// TIA Portal V20 export
// export: Created 2025-12-01T14:57:01.5792042Z, ExportSetting None, DisplayName Totally Integrated Automation Portal, DisplayVersion V20 Update 3, DisplayName TIA Portal Openness, DisplayVersion V20 Update 3, DisplayName TIA Portal Version Control Interface, DisplayVersion V20 Update 3, DisplayName STEP 7 Professional, DisplayVersion V20 Update 3, DisplayName STEP 7 Safety, DisplayVersion V20 Update 2, DisplayName WinCC Basic/Comfort/Advanced, DisplayVersion V20 Update 3, DisplayName WinCC Professional, DisplayVersion V20 Update 3, DisplayName WinCC Unified, DisplayVersion V20 Update 3
FUNCTION "FC458_TL_EMP_E1_S2_AUS" : Void   // FC458, LAD
{ S7_Optimized_Access := 'FALSE' }
AUTHOR : TLigero
NAME : 20160208
VERSION : 3.5
// stored: AutoNumber false, SetENOAutomatically false
   VAR_INPUT
      Mesa : UInt;
      En_Tension : Bool;
      phsMx_E1 : Bool;
      Termico_E1_Tx : Bool;
      Avance_E1_Tx_Ok : Bool;
      En_Emp_Recogido : Bool;
      En_Emp_Extendido : Bool;
      AVTF_MAnt_Mx : Bool;
      PTF_Mx_MSig : Bool;
      NXT_Avance : Bool;
      V_CNT_ApHsMx_E1 : UDInt;
      V_Paro : UDInt;
      V_Emp_Sacado : UDInt;
      V_TOut_Empujador : UDInt;
      V_TOut_Tx_Mx : UDInt;
   END_VAR
   VAR_OUTPUT
      PTF_MAnt_Mx : Bool;
      AVTF_Mx_MSig : Bool;
      NXT_Descarga_Act : Bool;
   END_VAR
   VAR_IN_OUT
      Mem_Aux_FNE1 : Bool;
      Mem_FN_phs_E1 : Bool;
      Mem_Aux_FNS2 : Bool;
      Mem_FN_phs_S2 : Bool;
      Mem_Flanco_Recog : Bool;
   END_VAR
   VAR_TEMP
      Mem_CNT_Aus_Ent : Bool;
      Temp_Emp_Sacado : Bool;
      Aux_Parar : Bool;
      tout_atasco : Bool;
      Tout_Empujador : Bool;
      Mem_CNT_Tmp_Paro_Tx : Bool;
      TEMP_MA_TR_Pos_E1 : Bool;
      TEMP_MA_TR_Pos_S2 : Bool;
      ok_tension : Bool;
   END_VAR
   VAR_TEMP   // added for the SCL form of the ladder/FBD networks
      _w1 : Bool;
      _w2 : Bool;
   END_VAR
BEGIN

REGION Network 1: Marca General Error
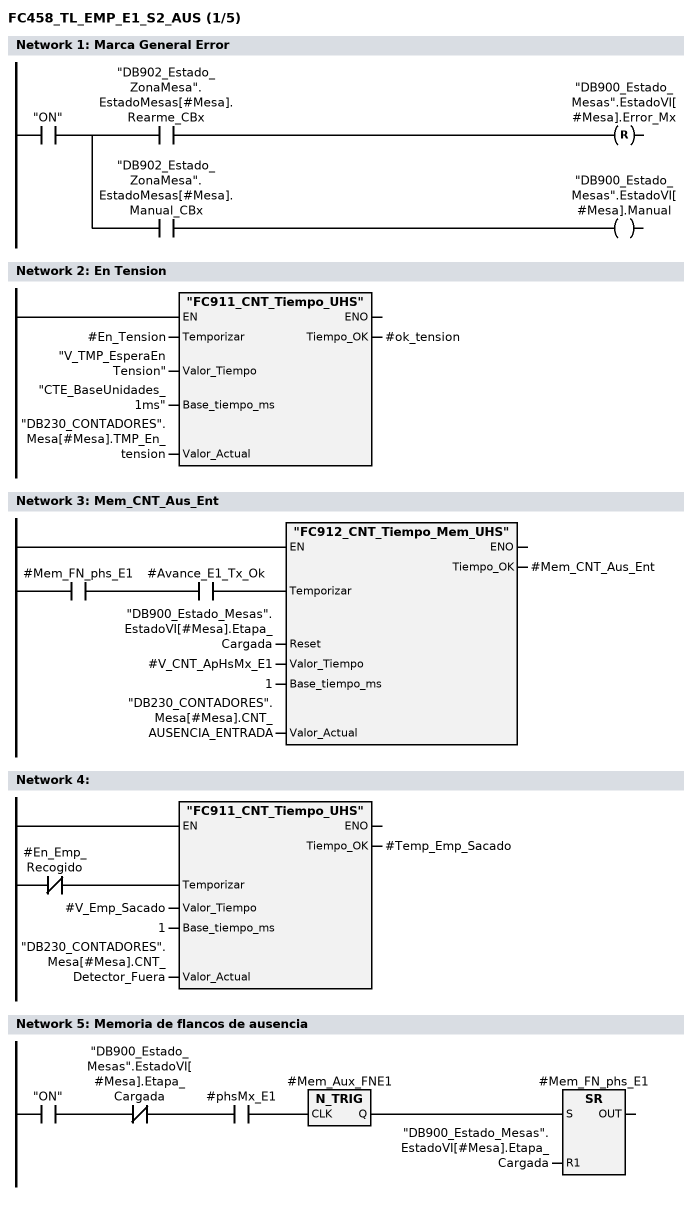
   RUNG wire#powerrail
      Contact( "ON" )
      wire#w1
      Contact( "DB902_Estado_ZonaMesa".EstadoMesas[#Mesa].Rearme_CBx )
      R_Coil( "DB900_Estado_Mesas".EstadoVI[#Mesa].Error_Mx )
   END_RUNG
   RUNG wire#w1
      Contact( "DB902_Estado_ZonaMesa".EstadoMesas[#Mesa].Manual_CBx )
      Coil( "DB900_Estado_Mesas".EstadoVI[#Mesa].Manual )
   END_RUNG
   // the same network as SCL:
   IF "ON" AND "DB902_Estado_ZonaMesa".EstadoMesas[#Mesa].Rearme_CBx THEN
       "DB900_Estado_Mesas".EstadoVI[#Mesa].Error_Mx := FALSE;
   END_IF;
   "DB900_Estado_Mesas".EstadoVI[#Mesa].Manual := "ON" AND "DB902_Estado_ZonaMesa".EstadoMesas[#Mesa].Manual_CBx;
END_REGION

REGION Network 2: En Tension
   RUNG wire#powerrail
      "FC911_CNT_Tiempo_UHS"(Temporizar := #En_Tension, Valor_Tiempo := "V_TMP_EsperaEnTension", Base_tiempo_ms := "CTE_BaseUnidades_1ms", Valor_Actual := "DB230_CONTADORES".Mesa[#Mesa].TMP_En_tension, Tiempo_OK => #ok_tension)
   END_RUNG
   // the same network as SCL:
   "FC911_CNT_Tiempo_UHS"(Temporizar := #En_Tension,
                          Valor_Tiempo := "V_TMP_EsperaEnTension",
                          Base_tiempo_ms := "CTE_BaseUnidades_1ms",
                          Valor_Actual := "DB230_CONTADORES".Mesa[#Mesa].TMP_En_tension,
                          Tiempo_OK => #ok_tension);
END_REGION

REGION Network 3: Mem_CNT_Aus_Ent
   RUNG wire#powerrail
      "FC912_CNT_Tiempo_Mem_UHS"(Temporizar := wire#w1, Reset := "DB900_Estado_Mesas".EstadoVI[#Mesa].Etapa_Cargada, Valor_Tiempo := #V_CNT_ApHsMx_E1, Base_tiempo_ms := 1, Valor_Actual := "DB230_CONTADORES".Mesa[#Mesa].CNT_AUSENCIA_ENTRADA, Tiempo_OK => #Mem_CNT_Aus_Ent)
   END_RUNG
   RUNG wire#powerrail
      Contact( #Mem_FN_phs_E1 )
      Contact( #Avance_E1_Tx_Ok )
   END_RUNG wire#w1
   // the same network as SCL:
   "FC912_CNT_Tiempo_Mem_UHS"(Temporizar := #Mem_FN_phs_E1 AND #Avance_E1_Tx_Ok,
                           Reset := "DB900_Estado_Mesas".EstadoVI[#Mesa].Etapa_Cargada,
                           Valor_Tiempo := #V_CNT_ApHsMx_E1,
                           Base_tiempo_ms := 1,
                           Valor_Actual := "DB230_CONTADORES".Mesa[#Mesa].CNT_AUSENCIA_ENTRADA,
                           Tiempo_OK => #Mem_CNT_Aus_Ent);
END_REGION

REGION Network 4
   RUNG wire#powerrail
      "FC911_CNT_Tiempo_UHS"(Temporizar := wire#w1, Valor_Tiempo := #V_Emp_Sacado, Base_tiempo_ms := 1, Valor_Actual := "DB230_CONTADORES".Mesa[#Mesa].CNT_Detector_Fuera, Tiempo_OK => #Temp_Emp_Sacado)
   END_RUNG
   RUNG wire#powerrail
      I_Contact( #En_Emp_Recogido )
   END_RUNG wire#w1
   // the same network as SCL:
   "FC911_CNT_Tiempo_UHS"(Temporizar := NOT #En_Emp_Recogido,
                          Valor_Tiempo := #V_Emp_Sacado,
                          Base_tiempo_ms := 1,
                          Valor_Actual := "DB230_CONTADORES".Mesa[#Mesa].CNT_Detector_Fuera,
                          Tiempo_OK => #Temp_Emp_Sacado);
END_REGION

REGION Network 5: Memoria de flancos de ausencia
   RUNG wire#powerrail
      Contact( "ON" )
      I_Contact( "DB900_Estado_Mesas".EstadoVI[#Mesa].Etapa_Cargada )
      Contact( #phsMx_E1 )
      N_Trig( #Mem_Aux_FNE1 )
      S_SR(operand := #Mem_FN_phs_E1, r1 := "DB900_Estado_Mesas".EstadoVI[#Mesa].Etapa_Cargada)
   END_RUNG
   // the same network as SCL:
   #_w1 := "ON" AND NOT "DB900_Estado_Mesas".EstadoVI[#Mesa].Etapa_Cargada AND #phsMx_E1;
   #_w2 := NOT #_w1 AND #Mem_Aux_FNE1;   // falling edge
   #Mem_Aux_FNE1 := #_w1;
   IF #_w2 THEN
       #Mem_FN_phs_E1 := TRUE;   // SR flip-flop
   END_IF;
   IF "DB900_Estado_Mesas".EstadoVI[#Mesa].Etapa_Cargada THEN #Mem_FN_phs_E1 := FALSE; END_IF;
END_REGION

REGION Network 6: PARO
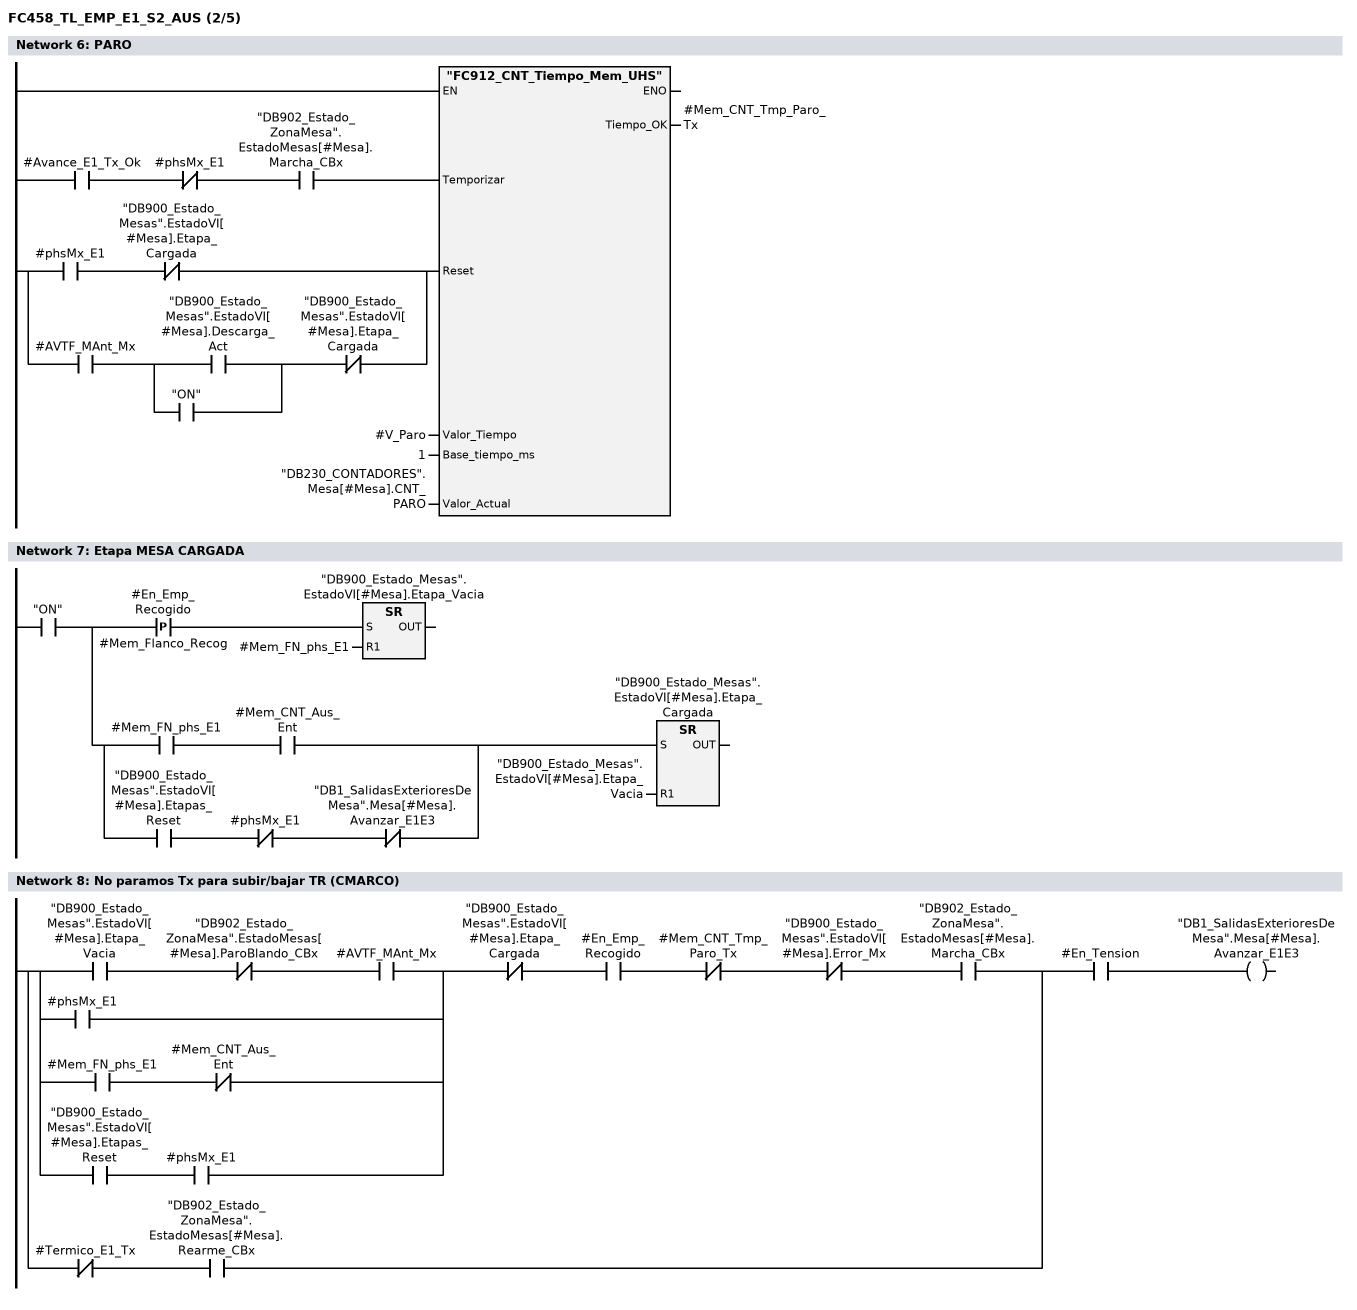
   RUNG wire#powerrail
      "FC912_CNT_Tiempo_Mem_UHS"(Temporizar := wire#w1, Reset := wire#w4, Valor_Tiempo := #V_Paro, Base_tiempo_ms := 1, Valor_Actual := "DB230_CONTADORES".Mesa[#Mesa].CNT_PARO, Tiempo_OK => #Mem_CNT_Tmp_Paro_Tx)
   END_RUNG
   RUNG wire#powerrail
      Contact( #Avance_E1_Tx_Ok )
      I_Contact( #phsMx_E1 )
      Contact( "DB902_Estado_ZonaMesa".EstadoMesas[#Mesa].Marcha_CBx )
   END_RUNG wire#w1
   RUNG wire#powerrail
      Contact( #phsMx_E1 )
      I_Contact( "DB900_Estado_Mesas".EstadoVI[#Mesa].Etapa_Cargada )
   END_RUNG wire#w4
   RUNG wire#powerrail
      Contact( #AVTF_MAnt_Mx )
      wire#w2
      Contact( "DB900_Estado_Mesas".EstadoVI[#Mesa].Descarga_Act )
      wire#w3
      I_Contact( "DB900_Estado_Mesas".EstadoVI[#Mesa].Etapa_Cargada )
   END_RUNG wire#w4
   RUNG wire#w2
      Contact( "ON" )
   END_RUNG wire#w3
   // the same network as SCL:
   "FC912_CNT_Tiempo_Mem_UHS"(Temporizar := #Avance_E1_Tx_Ok AND NOT #phsMx_E1 AND "DB902_Estado_ZonaMesa".EstadoMesas[#Mesa].Marcha_CBx,
                           Reset := (#phsMx_E1 AND NOT "DB900_Estado_Mesas".EstadoVI[#Mesa].Etapa_Cargada) OR (#AVTF_MAnt_Mx AND ("DB900_Estado_Mesas".EstadoVI[#Mesa].Descarga_Act OR "ON") AND NOT "DB900_Estado_Mesas".EstadoVI[#Mesa].Etapa_Cargada),
                           Valor_Tiempo := #V_Paro,
                           Base_tiempo_ms := 1,
                           Valor_Actual := "DB230_CONTADORES".Mesa[#Mesa].CNT_PARO,
                           Tiempo_OK => #Mem_CNT_Tmp_Paro_Tx);
END_REGION

REGION Network 7: Etapa MESA CARGADA
   RUNG wire#powerrail
      Contact( "ON" )
      wire#w1
      P_Contact(operand := #En_Emp_Recogido, bit := #Mem_Flanco_Recog)
      S_SR(operand := "DB900_Estado_Mesas".EstadoVI[#Mesa].Etapa_Vacia, r1 := #Mem_FN_phs_E1)
   END_RUNG
   RUNG wire#w1
      Contact( #Mem_FN_phs_E1 )
      Contact( #Mem_CNT_Aus_Ent )
      wire#w2
      S_SR(operand := "DB900_Estado_Mesas".EstadoVI[#Mesa].Etapa_Cargada, r1 := "DB900_Estado_Mesas".EstadoVI[#Mesa].Etapa_Vacia)
   END_RUNG
   RUNG wire#w1
      Contact( "DB900_Estado_Mesas".EstadoVI[#Mesa].Etapas_Reset )
      I_Contact( #phsMx_E1 )
      I_Contact( "DB1_SalidasExterioresDeMesa".Mesa[#Mesa].Avanzar_E1E3 )
   END_RUNG wire#w2
   // the same network as SCL:
   #_w1 := "ON" AND #En_Emp_Recogido AND NOT #Mem_Flanco_Recog;   // rising edge of #En_Emp_Recogido
   #Mem_Flanco_Recog := #En_Emp_Recogido;
   IF #_w1 THEN
       "DB900_Estado_Mesas".EstadoVI[#Mesa].Etapa_Vacia := TRUE;   // SR flip-flop
   END_IF;
   IF #Mem_FN_phs_E1 THEN "DB900_Estado_Mesas".EstadoVI[#Mesa].Etapa_Vacia := FALSE; END_IF;
   #_w2 := "DB900_Estado_Mesas".EstadoVI[#Mesa].Etapa_Vacia;
   IF "ON" AND ((#Mem_FN_phs_E1 AND #Mem_CNT_Aus_Ent) OR ("DB900_Estado_Mesas".EstadoVI[#Mesa].Etapas_Reset AND NOT #phsMx_E1 AND NOT "DB1_SalidasExterioresDeMesa".Mesa[#Mesa].Avanzar_E1E3)) THEN
       "DB900_Estado_Mesas".EstadoVI[#Mesa].Etapa_Cargada := TRUE;   // SR flip-flop
   END_IF;
   IF #_w2 THEN "DB900_Estado_Mesas".EstadoVI[#Mesa].Etapa_Cargada := FALSE; END_IF;
END_REGION

REGION Network 8: No paramos Tx para subir/bajar TR (CMARCO)
   RUNG wire#powerrail
      Contact( "DB900_Estado_Mesas".EstadoVI[#Mesa].Etapa_Vacia )
      I_Contact( "DB902_Estado_ZonaMesa".EstadoMesas[#Mesa].ParoBlando_CBx )
      Contact( #AVTF_MAnt_Mx )
      wire#w1
      I_Contact( "DB900_Estado_Mesas".EstadoVI[#Mesa].Etapa_Cargada )
      Contact( #En_Emp_Recogido )
      I_Contact( #Mem_CNT_Tmp_Paro_Tx )
      I_Contact( "DB900_Estado_Mesas".EstadoVI[#Mesa].Error_Mx )
      Contact( "DB902_Estado_ZonaMesa".EstadoMesas[#Mesa].Marcha_CBx )
      wire#w2
      Contact( #En_Tension )
      Coil( "DB1_SalidasExterioresDeMesa".Mesa[#Mesa].Avanzar_E1E3 )
   END_RUNG
   RUNG wire#powerrail
      Contact( #phsMx_E1 )
   END_RUNG wire#w1
   RUNG wire#powerrail
      Contact( #Mem_FN_phs_E1 )
      I_Contact( #Mem_CNT_Aus_Ent )
   END_RUNG wire#w1
   RUNG wire#powerrail
      Contact( "DB900_Estado_Mesas".EstadoVI[#Mesa].Etapas_Reset )
      Contact( #phsMx_E1 )
   END_RUNG wire#w1
   RUNG wire#powerrail
      I_Contact( #Termico_E1_Tx )
      Contact( "DB902_Estado_ZonaMesa".EstadoMesas[#Mesa].Rearme_CBx )
   END_RUNG wire#w2
   // the same network as SCL:
   "DB1_SalidasExterioresDeMesa".Mesa[#Mesa].Avanzar_E1E3 := (((("DB900_Estado_Mesas".EstadoVI[#Mesa].Etapa_Vacia AND NOT "DB902_Estado_ZonaMesa".EstadoMesas[#Mesa].ParoBlando_CBx AND #AVTF_MAnt_Mx) OR #phsMx_E1 OR (#Mem_FN_phs_E1 AND NOT #Mem_CNT_Aus_Ent) OR ("DB900_Estado_Mesas".EstadoVI[#Mesa].Etapas_Reset AND #phsMx_E1)) AND NOT "DB900_Estado_Mesas".EstadoVI[#Mesa].Etapa_Cargada AND #En_Emp_Recogido AND NOT #Mem_CNT_Tmp_Paro_Tx AND NOT "DB900_Estado_Mesas".EstadoVI[#Mesa].Error_Mx AND "DB902_Estado_ZonaMesa".EstadoMesas[#Mesa].Marcha_CBx) OR (NOT #Termico_E1_Tx AND "DB902_Estado_ZonaMesa".EstadoMesas[#Mesa].Rearme_CBx)) AND #En_Tension;
END_REGION

REGION Network 9: Aviso mesa siguiente
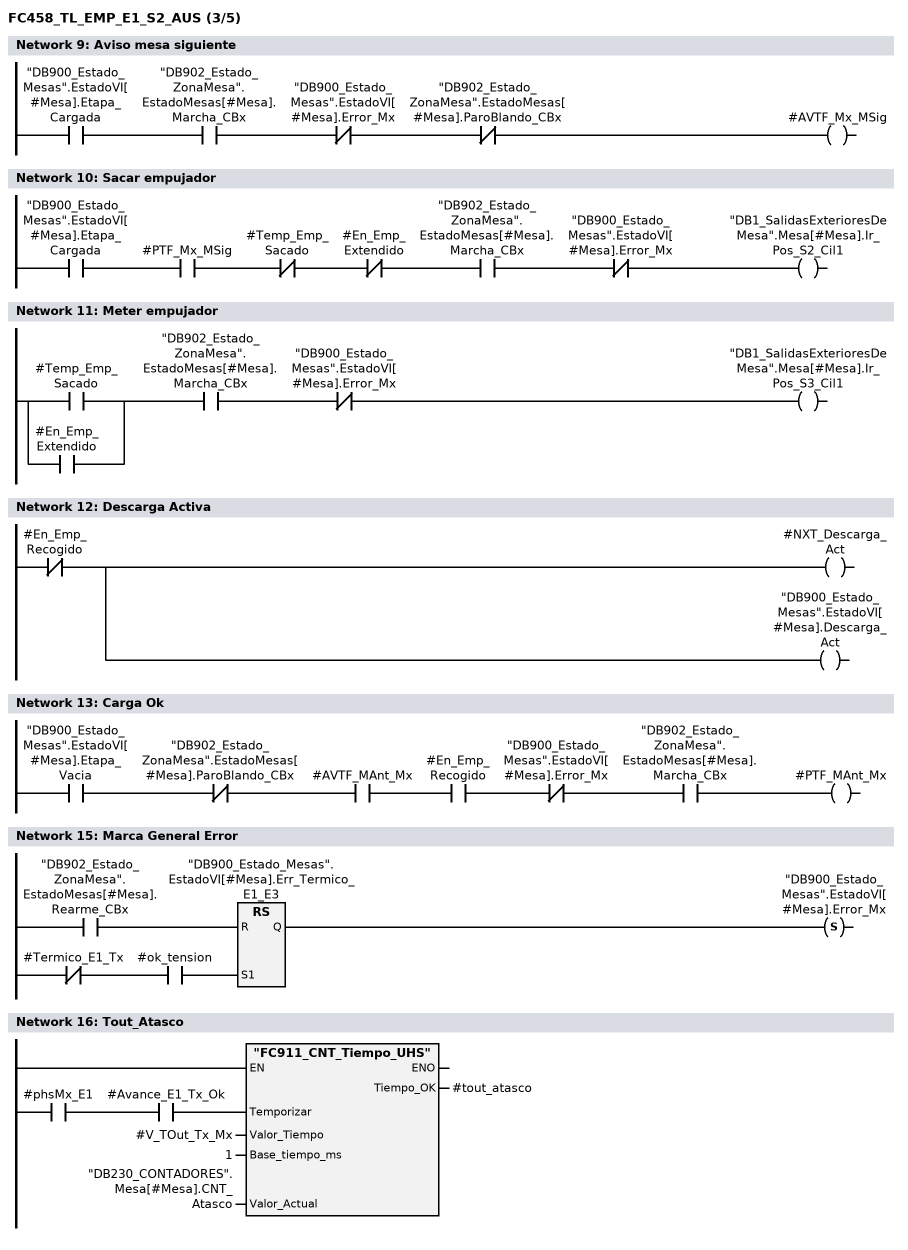
   RUNG wire#powerrail
      Contact( "DB900_Estado_Mesas".EstadoVI[#Mesa].Etapa_Cargada )
      Contact( "DB902_Estado_ZonaMesa".EstadoMesas[#Mesa].Marcha_CBx )
      I_Contact( "DB900_Estado_Mesas".EstadoVI[#Mesa].Error_Mx )
      I_Contact( "DB902_Estado_ZonaMesa".EstadoMesas[#Mesa].ParoBlando_CBx )
      Coil( #AVTF_Mx_MSig )
   END_RUNG
   // the same network as SCL:
   #AVTF_Mx_MSig := "DB900_Estado_Mesas".EstadoVI[#Mesa].Etapa_Cargada AND "DB902_Estado_ZonaMesa".EstadoMesas[#Mesa].Marcha_CBx AND NOT "DB900_Estado_Mesas".EstadoVI[#Mesa].Error_Mx AND NOT "DB902_Estado_ZonaMesa".EstadoMesas[#Mesa].ParoBlando_CBx;
END_REGION

REGION Network 10: Sacar empujador
   RUNG wire#powerrail
      Contact( "DB900_Estado_Mesas".EstadoVI[#Mesa].Etapa_Cargada )
      Contact( #PTF_Mx_MSig )
      I_Contact( #Temp_Emp_Sacado )
      I_Contact( #En_Emp_Extendido )
      Contact( "DB902_Estado_ZonaMesa".EstadoMesas[#Mesa].Marcha_CBx )
      I_Contact( "DB900_Estado_Mesas".EstadoVI[#Mesa].Error_Mx )
      Coil( "DB1_SalidasExterioresDeMesa".Mesa[#Mesa].Ir_Pos_S2_Cil1 )
   END_RUNG
   // the same network as SCL:
   "DB1_SalidasExterioresDeMesa".Mesa[#Mesa].Ir_Pos_S2_Cil1 := "DB900_Estado_Mesas".EstadoVI[#Mesa].Etapa_Cargada AND #PTF_Mx_MSig AND NOT #Temp_Emp_Sacado AND NOT #En_Emp_Extendido AND "DB902_Estado_ZonaMesa".EstadoMesas[#Mesa].Marcha_CBx AND NOT "DB900_Estado_Mesas".EstadoVI[#Mesa].Error_Mx;
END_REGION

REGION Network 11: Meter empujador
   RUNG wire#powerrail
      Contact( #Temp_Emp_Sacado )
      wire#w1
      Contact( "DB902_Estado_ZonaMesa".EstadoMesas[#Mesa].Marcha_CBx )
      I_Contact( "DB900_Estado_Mesas".EstadoVI[#Mesa].Error_Mx )
      Coil( "DB1_SalidasExterioresDeMesa".Mesa[#Mesa].Ir_Pos_S3_Cil1 )
   END_RUNG
   RUNG wire#powerrail
      Contact( #En_Emp_Extendido )
   END_RUNG wire#w1
   // the same network as SCL:
   "DB1_SalidasExterioresDeMesa".Mesa[#Mesa].Ir_Pos_S3_Cil1 := (#Temp_Emp_Sacado OR #En_Emp_Extendido) AND "DB902_Estado_ZonaMesa".EstadoMesas[#Mesa].Marcha_CBx AND NOT "DB900_Estado_Mesas".EstadoVI[#Mesa].Error_Mx;
END_REGION

REGION Network 12: Descarga Activa
   RUNG wire#powerrail
      I_Contact( #En_Emp_Recogido )
      wire#w1
      Coil( #NXT_Descarga_Act )
   END_RUNG
   RUNG wire#w1
      Coil( "DB900_Estado_Mesas".EstadoVI[#Mesa].Descarga_Act )
   END_RUNG
   // the same network as SCL:
   #NXT_Descarga_Act := NOT #En_Emp_Recogido;
   "DB900_Estado_Mesas".EstadoVI[#Mesa].Descarga_Act := NOT #En_Emp_Recogido;
END_REGION

REGION Network 13: Carga Ok
   RUNG wire#powerrail
      Contact( "DB900_Estado_Mesas".EstadoVI[#Mesa].Etapa_Vacia )
      I_Contact( "DB902_Estado_ZonaMesa".EstadoMesas[#Mesa].ParoBlando_CBx )
      Contact( #AVTF_MAnt_Mx )
      Contact( #En_Emp_Recogido )
      I_Contact( "DB900_Estado_Mesas".EstadoVI[#Mesa].Error_Mx )
      Contact( "DB902_Estado_ZonaMesa".EstadoMesas[#Mesa].Marcha_CBx )
      Coil( #PTF_MAnt_Mx )
   END_RUNG
   // the same network as SCL:
   #PTF_MAnt_Mx := "DB900_Estado_Mesas".EstadoVI[#Mesa].Etapa_Vacia AND NOT "DB902_Estado_ZonaMesa".EstadoMesas[#Mesa].ParoBlando_CBx AND #AVTF_MAnt_Mx AND #En_Emp_Recogido AND NOT "DB900_Estado_Mesas".EstadoVI[#Mesa].Error_Mx AND "DB902_Estado_ZonaMesa".EstadoMesas[#Mesa].Marcha_CBx;
END_REGION

REGION Network 14: Extender empujador
END_REGION

REGION Network 15: Marca General Error
   RUNG wire#powerrail
      Contact( "DB902_Estado_ZonaMesa".EstadoMesas[#Mesa].Rearme_CBx )
      S_RS(operand := "DB900_Estado_Mesas".EstadoVI[#Mesa].Err_Termico_E1_E3, s1 := wire#w1)
      S_Coil( "DB900_Estado_Mesas".EstadoVI[#Mesa].Error_Mx )
   END_RUNG
   RUNG wire#powerrail
      I_Contact( #Termico_E1_Tx )
      Contact( #ok_tension )
   END_RUNG wire#w1
   // the same network as SCL:
   IF "DB902_Estado_ZonaMesa".EstadoMesas[#Mesa].Rearme_CBx THEN
       "DB900_Estado_Mesas".EstadoVI[#Mesa].Err_Termico_E1_E3 := FALSE;   // RS flip-flop
   END_IF;
   IF NOT #Termico_E1_Tx AND #ok_tension THEN
       "DB900_Estado_Mesas".EstadoVI[#Mesa].Err_Termico_E1_E3 := TRUE;
   END_IF;
   IF "DB900_Estado_Mesas".EstadoVI[#Mesa].Err_Termico_E1_E3 THEN
       "DB900_Estado_Mesas".EstadoVI[#Mesa].Error_Mx := TRUE;
   END_IF;
END_REGION

REGION Network 16: Tout_Atasco
   RUNG wire#powerrail
      "FC911_CNT_Tiempo_UHS"(Temporizar := wire#w1, Valor_Tiempo := #V_TOut_Tx_Mx, Base_tiempo_ms := 1, Valor_Actual := "DB230_CONTADORES".Mesa[#Mesa].CNT_Atasco, Tiempo_OK => #tout_atasco)
   END_RUNG
   RUNG wire#powerrail
      Contact( #phsMx_E1 )
      Contact( #Avance_E1_Tx_Ok )
   END_RUNG wire#w1
   // the same network as SCL:
   "FC911_CNT_Tiempo_UHS"(Temporizar := #phsMx_E1 AND #Avance_E1_Tx_Ok,
                          Valor_Tiempo := #V_TOut_Tx_Mx,
                          Base_tiempo_ms := 1,
                          Valor_Actual := "DB230_CONTADORES".Mesa[#Mesa].CNT_Atasco,
                          Tiempo_OK => #tout_atasco);
END_REGION

REGION Network 17: Error Tout avanuce E1E3
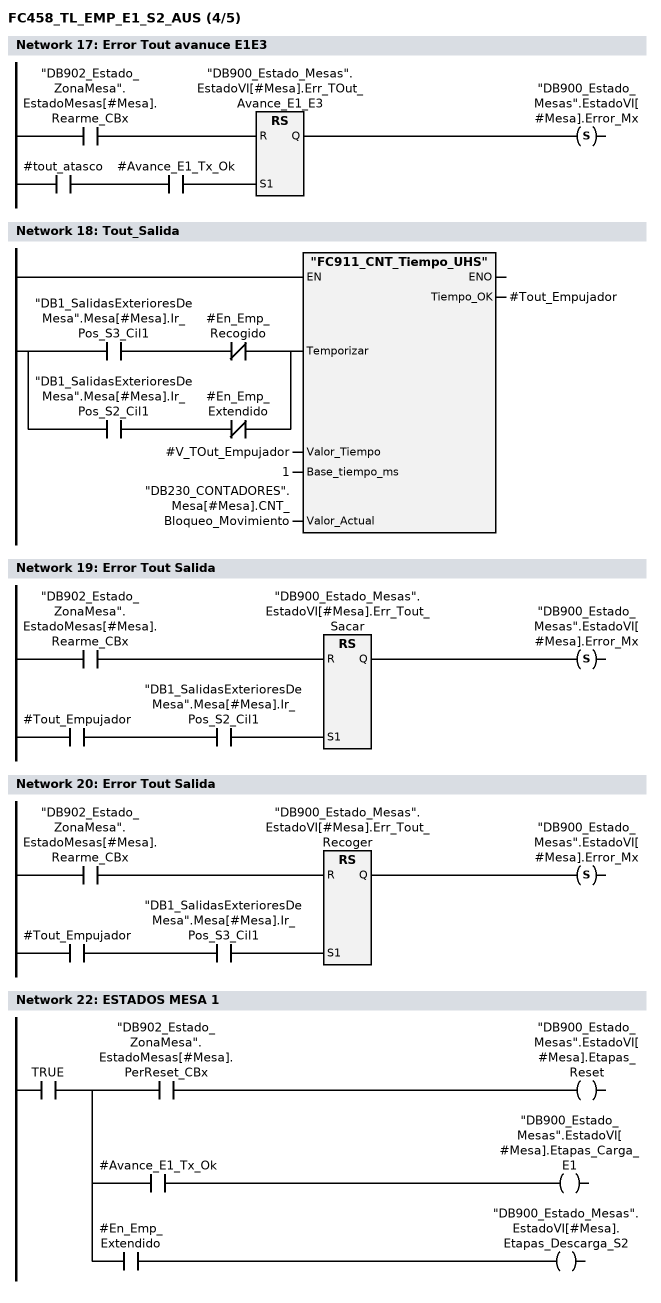
   RUNG wire#powerrail
      Contact( "DB902_Estado_ZonaMesa".EstadoMesas[#Mesa].Rearme_CBx )
      S_RS(operand := "DB900_Estado_Mesas".EstadoVI[#Mesa].Err_TOut_Avance_E1_E3, s1 := wire#w1)
      S_Coil( "DB900_Estado_Mesas".EstadoVI[#Mesa].Error_Mx )
   END_RUNG
   RUNG wire#powerrail
      Contact( #tout_atasco )
      Contact( #Avance_E1_Tx_Ok )
   END_RUNG wire#w1
   // the same network as SCL:
   IF "DB902_Estado_ZonaMesa".EstadoMesas[#Mesa].Rearme_CBx THEN
       "DB900_Estado_Mesas".EstadoVI[#Mesa].Err_TOut_Avance_E1_E3 := FALSE;   // RS flip-flop
   END_IF;
   IF #tout_atasco AND #Avance_E1_Tx_Ok THEN
       "DB900_Estado_Mesas".EstadoVI[#Mesa].Err_TOut_Avance_E1_E3 := TRUE;
   END_IF;
   IF "DB900_Estado_Mesas".EstadoVI[#Mesa].Err_TOut_Avance_E1_E3 THEN
       "DB900_Estado_Mesas".EstadoVI[#Mesa].Error_Mx := TRUE;
   END_IF;
END_REGION

REGION Network 18: Tout_Salida
   RUNG wire#powerrail
      "FC911_CNT_Tiempo_UHS"(Temporizar := wire#w1, Valor_Tiempo := #V_TOut_Empujador, Base_tiempo_ms := 1, Valor_Actual := "DB230_CONTADORES".Mesa[#Mesa].CNT_Bloqueo_Movimiento, Tiempo_OK => #Tout_Empujador)
   END_RUNG
   RUNG wire#powerrail
      Contact( "DB1_SalidasExterioresDeMesa".Mesa[#Mesa].Ir_Pos_S3_Cil1 )
      I_Contact( #En_Emp_Recogido )
   END_RUNG wire#w1
   RUNG wire#powerrail
      Contact( "DB1_SalidasExterioresDeMesa".Mesa[#Mesa].Ir_Pos_S2_Cil1 )
      I_Contact( #En_Emp_Extendido )
   END_RUNG wire#w1
   // the same network as SCL:
   "FC911_CNT_Tiempo_UHS"(Temporizar := ("DB1_SalidasExterioresDeMesa".Mesa[#Mesa].Ir_Pos_S3_Cil1 AND NOT #En_Emp_Recogido) OR ("DB1_SalidasExterioresDeMesa".Mesa[#Mesa].Ir_Pos_S2_Cil1 AND NOT #En_Emp_Extendido),
                          Valor_Tiempo := #V_TOut_Empujador,
                          Base_tiempo_ms := 1,
                          Valor_Actual := "DB230_CONTADORES".Mesa[#Mesa].CNT_Bloqueo_Movimiento,
                          Tiempo_OK => #Tout_Empujador);
END_REGION

REGION Network 19: Error Tout Salida
   RUNG wire#powerrail
      Contact( "DB902_Estado_ZonaMesa".EstadoMesas[#Mesa].Rearme_CBx )
      S_RS(operand := "DB900_Estado_Mesas".EstadoVI[#Mesa].Err_Tout_Sacar, s1 := wire#w1)
      S_Coil( "DB900_Estado_Mesas".EstadoVI[#Mesa].Error_Mx )
   END_RUNG
   RUNG wire#powerrail
      Contact( #Tout_Empujador )
      Contact( "DB1_SalidasExterioresDeMesa".Mesa[#Mesa].Ir_Pos_S2_Cil1 )
   END_RUNG wire#w1
   // the same network as SCL:
   #_w1 := #Tout_Empujador AND "DB1_SalidasExterioresDeMesa".Mesa[#Mesa].Ir_Pos_S2_Cil1;
   IF "DB902_Estado_ZonaMesa".EstadoMesas[#Mesa].Rearme_CBx THEN
       "DB900_Estado_Mesas".EstadoVI[#Mesa].Err_Tout_Sacar := FALSE;   // RS flip-flop
   END_IF;
   IF #_w1 THEN "DB900_Estado_Mesas".EstadoVI[#Mesa].Err_Tout_Sacar := TRUE; END_IF;
   IF "DB900_Estado_Mesas".EstadoVI[#Mesa].Err_Tout_Sacar THEN
       "DB900_Estado_Mesas".EstadoVI[#Mesa].Error_Mx := TRUE;
   END_IF;
END_REGION

REGION Network 20: Error Tout Salida
   RUNG wire#powerrail
      Contact( "DB902_Estado_ZonaMesa".EstadoMesas[#Mesa].Rearme_CBx )
      S_RS(operand := "DB900_Estado_Mesas".EstadoVI[#Mesa].Err_Tout_Recoger, s1 := wire#w1)
      S_Coil( "DB900_Estado_Mesas".EstadoVI[#Mesa].Error_Mx )
   END_RUNG
   RUNG wire#powerrail
      Contact( #Tout_Empujador )
      Contact( "DB1_SalidasExterioresDeMesa".Mesa[#Mesa].Ir_Pos_S3_Cil1 )
   END_RUNG wire#w1
   // the same network as SCL:
   #_w1 := #Tout_Empujador AND "DB1_SalidasExterioresDeMesa".Mesa[#Mesa].Ir_Pos_S3_Cil1;
   IF "DB902_Estado_ZonaMesa".EstadoMesas[#Mesa].Rearme_CBx THEN
       "DB900_Estado_Mesas".EstadoVI[#Mesa].Err_Tout_Recoger := FALSE;   // RS flip-flop
   END_IF;
   IF #_w1 THEN "DB900_Estado_Mesas".EstadoVI[#Mesa].Err_Tout_Recoger := TRUE; END_IF;
   IF "DB900_Estado_Mesas".EstadoVI[#Mesa].Err_Tout_Recoger THEN
       "DB900_Estado_Mesas".EstadoVI[#Mesa].Error_Mx := TRUE;
   END_IF;
END_REGION

REGION Network 22: ESTADOS MESA 1
   RUNG wire#powerrail
      Contact( TRUE )
      wire#w1
      Contact( "DB902_Estado_ZonaMesa".EstadoMesas[#Mesa].PerReset_CBx )
      Coil( "DB900_Estado_Mesas".EstadoVI[#Mesa].Etapas_Reset )
   END_RUNG
   RUNG wire#w1
      Contact( #Avance_E1_Tx_Ok )
      Coil( "DB900_Estado_Mesas".EstadoVI[#Mesa].Etapas_Carga_E1 )
   END_RUNG
   RUNG wire#w1
      Contact( #En_Emp_Extendido )
      Coil( "DB900_Estado_Mesas".EstadoVI[#Mesa].Etapas_Descarga_S2 )
   END_RUNG
   // the same network as SCL:
   "DB900_Estado_Mesas".EstadoVI[#Mesa].Etapas_Reset := TRUE AND "DB902_Estado_ZonaMesa".EstadoMesas[#Mesa].PerReset_CBx;
   "DB900_Estado_Mesas".EstadoVI[#Mesa].Etapas_Carga_E1 := TRUE AND #Avance_E1_Tx_Ok;
   "DB900_Estado_Mesas".EstadoVI[#Mesa].Etapas_Descarga_S2 := TRUE AND #En_Emp_Extendido;
END_REGION

REGION Network 23: Entradas Mesas
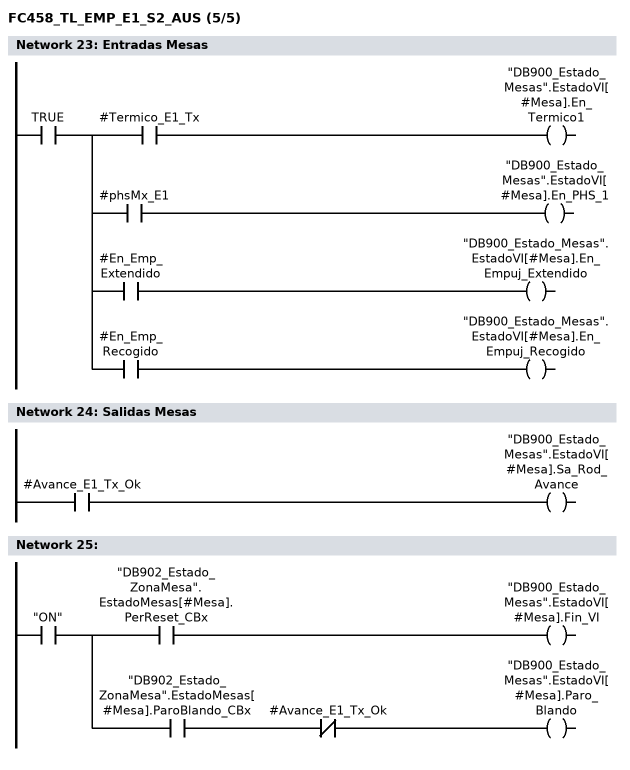
   RUNG wire#powerrail
      Contact( TRUE )
      wire#w1
      Contact( #Termico_E1_Tx )
      Coil( "DB900_Estado_Mesas".EstadoVI[#Mesa].En_Termico1 )
   END_RUNG
   RUNG wire#w1
      Contact( #phsMx_E1 )
      Coil( "DB900_Estado_Mesas".EstadoVI[#Mesa].En_PHS_1 )
   END_RUNG
   RUNG wire#w1
      Contact( #En_Emp_Extendido )
      Coil( "DB900_Estado_Mesas".EstadoVI[#Mesa].En_Empuj_Extendido )
   END_RUNG
   RUNG wire#w1
      Contact( #En_Emp_Recogido )
      Coil( "DB900_Estado_Mesas".EstadoVI[#Mesa].En_Empuj_Recogido )
   END_RUNG
   // the same network as SCL:
   "DB900_Estado_Mesas".EstadoVI[#Mesa].En_Termico1 := TRUE AND #Termico_E1_Tx;
   "DB900_Estado_Mesas".EstadoVI[#Mesa].En_PHS_1 := TRUE AND #phsMx_E1;
   "DB900_Estado_Mesas".EstadoVI[#Mesa].En_Empuj_Extendido := TRUE AND #En_Emp_Extendido;
   "DB900_Estado_Mesas".EstadoVI[#Mesa].En_Empuj_Recogido := TRUE AND #En_Emp_Recogido;
END_REGION

REGION Network 24: Salidas Mesas
   RUNG wire#powerrail
      Contact( #Avance_E1_Tx_Ok )
      Coil( "DB900_Estado_Mesas".EstadoVI[#Mesa].Sa_Rod_Avance )
   END_RUNG
   // the same network as SCL:
   "DB900_Estado_Mesas".EstadoVI[#Mesa].Sa_Rod_Avance := #Avance_E1_Tx_Ok;
END_REGION

REGION Network 25
   RUNG wire#powerrail
      Contact( "ON" )
      wire#w1
      Contact( "DB902_Estado_ZonaMesa".EstadoMesas[#Mesa].PerReset_CBx )
      Coil( "DB900_Estado_Mesas".EstadoVI[#Mesa].Fin_VI )
   END_RUNG
   RUNG wire#w1
      Contact( "DB902_Estado_ZonaMesa".EstadoMesas[#Mesa].ParoBlando_CBx )
      I_Contact( #Avance_E1_Tx_Ok )
      Coil( "DB900_Estado_Mesas".EstadoVI[#Mesa].Paro_Blando )
   END_RUNG
   // the same network as SCL:
   "DB900_Estado_Mesas".EstadoVI[#Mesa].Fin_VI := "ON" AND "DB902_Estado_ZonaMesa".EstadoMesas[#Mesa].PerReset_CBx;
   "DB900_Estado_Mesas".EstadoVI[#Mesa].Paro_Blando := "ON" AND "DB902_Estado_ZonaMesa".EstadoMesas[#Mesa].ParoBlando_CBx AND NOT #Avance_E1_Tx_Ok;
END_REGION
END_FUNCTION
